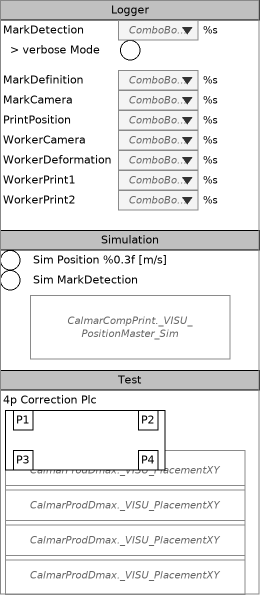
VISUALIZATION _VISU_Pm_Debug  // 260x595
VAR_IN_OUT
	mInst : FB_PrintModule_WEU;
END_VAR
    Rectangle (0,230 260x20), "Simulation"
    Ellipse (0,250 20x20), tooltip "Sim position"
        toggle mInst.fbPrintPosition._bSim
    Rectangle (30,250 200x20), "Sim Position %0.3f [m/s]", text variable: mInst.fbPrintPosition.fbPositionMaster._fSimSpeed
        OnMouseClick: write the text variable via Default
    Ellipse (0,270 20x20), tooltip "Sim position"
        toggle mInst.fbMarkDetection.bSimEnable
    Rectangle (30,270 200x20), "Sim MarkDetection"
    Rectangle (0,0 260x20), "Logger"
    Rectangle (0,20 120x20), "MarkDetection"
    Rectangle (0,70 120x20), "MarkDefinition"
    Rectangle (200,70 60x20), "%s", tooltip "LogLevel", text variable: mInst.fbMarkDefinition._loglevel
        OnMouseClick: write the text variable via Default
    Rectangle (0,90 120x20), "MarkCamera"
    Rectangle (200,90 60x20), "%s", tooltip "LogLevel", text variable: mInst.fbMarkCameraWeu._loglevel
        OnMouseClick: write the text variable via Default
    Rectangle (0,110 120x20), "PrintPosition"
    Rectangle (200,110 60x20), "%s", tooltip "LogLevel", text variable: mInst.fbPrintPosition._loglevel
        OnMouseClick: write the text variable via Default
    Rectangle (0,130 120x20), "WorkerCamera"
    Rectangle (200,130 60x20), "%s", tooltip "LogLevel", text variable: mInst.fbWorkerCamera._loglevel
        OnMouseClick: write the text variable via Default
    Rectangle (0,170 120x20), "WorkerPrint1"
    Rectangle (200,170 60x20), "%s", tooltip "LogLevel", text variable: mInst.fbWorkerPrint[1]._loglevel
        OnMouseClick: write the text variable via Default
    Rectangle (0,190 120x20), "WorkerPrint2"
    Rectangle (200,190 60x20), "%s", tooltip "LogLevel", text variable: mInst.fbWorkerPrint[2]._loglevel
        OnMouseClick: write the text variable via Default
    Rectangle (0,40 120x20), "> verbose Mode"
    Ellipse (120,40 20x20)
        toggle mInst.fbMarkDetection._bVerbose
    Rectangle (0,150 120x20), "WorkerDeformation"
    Rectangle (200,150 60x20), "%s", tooltip "LogLevel", text variable: mInst.fbWorkerDeformation._loglevel
        OnMouseClick: write the text variable via Default
    ComboBoxInteger (118,170 80x20), tooltip "LogLevel", variable: mInst.fbWorkerPrint[1]._loglevel, text list: 'LogSeverity'
    ComboBoxInteger (118,190 80x20), tooltip "LogLevel", variable: mInst.fbWorkerPrint[2]._loglevel, text list: 'LogSeverity'
    ComboBoxInteger (118,150 80x20), tooltip "LogLevel", variable: mInst.fbWorkerDeformation._loglevel, text list: 'LogSeverity'
    ComboBoxInteger (118,130 80x20), tooltip "LogLevel", variable: mInst.fbWorkerCamera._loglevel, text list: 'LogSeverity'
    ComboBoxInteger (118,110 80x20), tooltip "LogLevel", variable: mInst.fbPrintPosition._loglevel, text list: 'LogSeverity'
    ComboBoxInteger (118,90 80x20), tooltip "LogLevel", variable: mInst.fbMarkCameraWeu._loglevel, text list: 'LogSeverity'
    ComboBoxInteger (118,70 80x20), tooltip "LogLevel", variable: mInst.fbMarkDefinition._loglevel, text list: 'LogSeverity'
    Rectangle (200,20 60x20), "%s", tooltip "LogLevel", text variable: mInst.fbMarkDetection._loglevel
        OnMouseClick: write the text variable via Default
    ComboBoxInteger (118,20 80x20), tooltip "LogLevel", variable: mInst.fbMarkDetection._loglevel, text list: 'LogSeverity'
    Frame (30,295 200x64)
        shows CalmarCompPrint._VISU_PositionMaster_Sim(mInst := mInst.fbPrintPosition.fbPositionMaster)
    Frame (5,450 240x40)
        shows CalmarProdDmax._VISU_PlacementXY(m_Inst := mInst.fbFineAlignement._fbPUCorrPoints[1])
    Frame (5,485 240x40)
        shows CalmarProdDmax._VISU_PlacementXY(m_Inst := mInst.fbFineAlignement._fbPUCorrPoints[2])
    Frame (5,520 240x40)
        shows CalmarProdDmax._VISU_PlacementXY(m_Inst := mInst.fbFineAlignement._fbPUCorrPoints[3])
    Frame (5,555 240x40)
        shows CalmarProdDmax._VISU_PlacementXY(m_Inst := mInst.fbFineAlignement._fbPUCorrPoints[4])
    Rectangle (0,390 120x20), "4p Correction Plc"
    Group (5,410 69x30)
        RoundedRectangle (0,0 160x60)
        Rectangle (8,0 20x20), "P1"
        Rectangle (133,0 20x20), "P2"
        Rectangle (133,40 20x20), "P4"
        Rectangle (8,40 20x20), "P3"
    Rectangle (0,370 260x20), "Test"
END_VISUALIZATION

(* stored: Version 1.1.0.1, ProductVersion 3.1.4024.11
   Visu _VISU_Pm_Debug: Id {0aa3d8be-608b-4a72-b875-f5ae4d6aa908} *)
